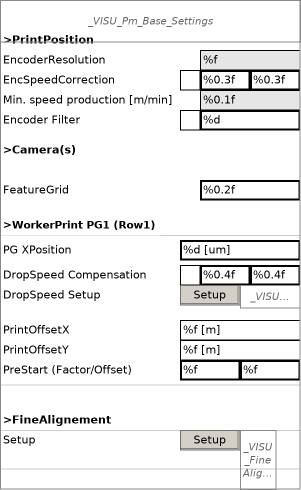
VISUALIZATION _VISU_Pm_Maxliner_Settings  // 301x490
VAR_IN_OUT
	mInst : FB_PrintModule_Maxliner;
END_VAR
    Rectangle (0,430 300x39)
    Rectangle (250,70 50x20), "%0.3f", tooltip "Encoder speed compensation reference speed", text variable: mInst.fbPrintPosition._fSpeedCompRefSpeed
        OnMouseClick: write the text variable via Default
    Rectangle (200,70 50x20), "%0.3f", tooltip "Encoder speed compensation factor", text variable: mInst.fbPrintPosition._fSpeedCompFactor
        OnMouseClick: write the text variable via Default
    RoundedRectangle (180,70 20x20)
        toggle mInst.fbPrintPosition._bEnSpeedComp
    Rectangle (0,70 180x20), "EncSpeedCorrection"
    Rectangle (0,50 180x20), "EncoderResolution"
    Rectangle (200,50 100x20), "%f", tooltip "by calculation", text variable: mInst.fbPrintPosition._fEncoderResolution
    Rectangle (0,235 300x150)
    Rectangle (0,265 180x20), "DropSpeed Compensation"
    Rectangle (200,265 50x20), "%0.4f", tooltip "DropSpeed [m/s]", text variable: mInst.fbWorkerPrint[1].fbDropSpeedComp.fDropSpeed
        OnMouseClick: write the text variable via Default
    Rectangle (250,265 50x20), "%0.4f", tooltip "Dead/Add Time [ms]", text variable: mInst.fbWorkerPrint[1].fbDropSpeedComp.fDropSpeedDeadTime
        OnMouseClick: write the text variable via Default
    RoundedRectangle (180,265 20x20), tooltip "Enabled compensation", input disabled if: TRUE
        toggle mInst.fbWorkerPrint[1].fbDropSpeedComp._bEnable p2164770859=TRUE
    Button (180,285 60x20), "Setup", tooltip "Setup"
        toggle mInst.fbWorkerPrint[1].bShowDropSpeedSetup
    Rectangle (0,285 180x20), "DropSpeed Setup"
    Rectangle (0,30 180x20), ">PrintPosition"
    Rectangle (0,90 180x20), "Min. speed production [m/min]"
    Rectangle (200,90 100x20), "%0.1f", tooltip "constant", text variable: mInst.fC_MinimalProductionSpeed_in_MpMin
    Rectangle (0,140 180x20), ">Camera(s)"
    Rectangle (200,110 100x20), "%d", tooltip "Filter depth", text variable: mInst.fbPrintPosition.fbPositionMaster.nFilterDepth
        OnMouseClick: write the text variable via Default
    RoundedRectangle (180,110 20x20)
        toggle mInst.fbPrintPosition.fbPositionMaster.bEnableFilter
    Rectangle (0,110 180x20), "Encoder Filter"
    Rectangle (0,180 180x20), "FeatureGrid"
    Rectangle (200,180 100x20), "%0.2f", text variable: mInst.fbWorkerCamera._fFeatureGrid
        OnMouseDown: write the text variable via Default
    Rectangle (0,410 180x20), ">FineAlignement"
    Button (180,430 60x20), "Setup", tooltip "Setup"
        toggle minst.fbView.bShowFineAlignement
    Rectangle (0,430 180x20), "Setup"
    Frame (0,0 301x42)
        shows _VISU_Pm_Base_Settings(mInst := mInst)
    Rectangle (0,320 180x20), "PrintOffsetX"
    Rectangle (0,340 180x20), "PrintOffsetY"
    Rectangle (180,320 120x20), "%f [m]", text variable: mInst.fbWorkerPrint[1].fPrintStartOffset, input disabled if: TRUE
    Rectangle (180,340 120x20), "%f [m]", text variable: mInst.fbWorkerPrint[1].fPrintYOffset, input disabled if: TRUE
    Rectangle (0,215 160x20), ">WorkerPrint PG1 (Row1)"
    Rectangle (0,240 180x20), "PG XPosition"
    Rectangle (180,240 120x20), "%d [um]", text variable: mInst.fbAdsPg[1].stAds.sI_ShiftPositionX.lI_Val
        OnMouseClick: write the text variable via Default
    Rectangle (0,360 180x20), "PreStart (Factor/Offset)"
    Rectangle (180,360 60x20), "%f", tooltip "PreStart ShiftFactor", text variable: mInst.fbWorkerPrint[1]._fStartShiftFactor
        OnMouseClick: write the text variable via Default
    Rectangle (240,360 60x20), "%f", tooltip "PreStart ShiftOffset", text variable: mInst.fbWorkerPrint[1]._fStartShiftOffset
        OnMouseClick: write the text variable via Default
    Frame (240,285 60x23), invisible if: NOT mInst.fbWorkerPrint[1].bShowDropSpeedSetup
        shows _VISU_DropSpeedComp_Setup(mInst := mInst.fbWorkerPrint[1].fbDropSpeedComp)
    Frame (240,430 36x60), invisible if: NOT minst.fbView.bShowFineAlignement
        shows _VISU_FineAlignment(mInst := mInst.fbFineAlignement)
END_VISUALIZATION

(* stored: Version 1.1.0.1, ProductVersion 3.1.4024.11
   Visu _VISU_Pm_Maxliner_Settings: Id {836ce0fa-7bc2-4109-b1d5-e7b08564c28a} *)
